# EPICS substitutions: apps/cRioApp/Db/gas_cRIO_BONUS_intlk.substitutions
file "db/mmIntlk.template" {
pattern { P R PV LOW HIGH CTRL CTRLVAL PREC DESC }
{ B_BONUS_INTLK_ Flow         B_BONUS_GAS_MFC_Flow          B_BONUS_GAS_MFC_Flow.LOLO          B_BONUS_GAS_MFC_Flow.HIHI          B_BONUS_HV:off 1 2 "HV Off if Flow LOLO/HIHI" }
{ B_BONUS_INTLK_ FlowSetDiff  B_BONUS_GAS_MFC_Flow:watchdog B_BONUS_GAS_MFC_Flow:watchdog.LOLO B_BONUS_GAS_MFC_Flow:watchdog.HIHI B_BONUS_HV:off 1 2 "HV Off if Flow-FlowSet LOLO/HIHI" }
{ B_BONUS_INTLK_ RTPC_Press   B_BONUS_RTPC_Press            B_BONUS_RTPC_Press.LOLO            B_BONUS_RTPC_Press.HIHI            B_BONUS_HV:off 1 2 "HV Off if RTPC Pressure LOLO/HIHI" }
{ B_BONUS_INTLK_ Diff_Press   B_BONUS_GAS_DP                B_BONUS_GAS_DP.LOLO                B_BONUS_GAS_DP.HIHI                B_BONUS_HV:off 1 2 "HV Off if Diff. Pressure LOLO/HIHI" }
{ B_BONUS_INTLK_ Buffer_Press B_BONUS_GAS_He_Buffer_Press   B_BONUS_GAS_He_Buffer_Press.LOLO   B_BONUS_GAS_He_Buffer_Press.HIHI   B_BONUS_HV:off 1 2 "HV Off if He Buffer Pressure LOLO/HIHI" }
}
